FUNCTION_BLOCK FB_Double_drum
VAR_INPUT
	Lh_raw_depth:REAL; (*Raw left hand drum depth*)
	Rh_raw_depth:REAL; (*Raw right hand drum depth*)
	Lh_speed:REAL; (*Left drum speed in mm/s*)
	Rh_speed:REAL; (*Right drum speed in mm/s*)
	Tacho_speed:REAL; (*Tacho speed in mm/s*)
	Speed_ref:REAL; (*Speed reference output to drive in mm/s*)
	Lh_going_up:BOOL; (*Left conveyance moving in the upward direction (forward)*)
	Rh_going_up:BOOL; (*Right conveyance moving in the upward direction (forward)*)
	Lh_movement:BOOL; (*Movement detected on left drum since the brakes were last applied*)
	Rh_movement:BOOL; (*Movement detected on right drum since the brakes were last applied*)
	Enc_xcheck_dist:REAL; (*Allowed variation in the sum of the left and right raw depths since both clutches were put in or a winder reset*)
	Tacho_xcheck_abs:REAL; (*Allowed absolute difference between the tacho speed and encoder speed (added to Tacho_xcheck_percent)*)
	Tacho_xcheck_percent:REAL; (*Allowed percentage difference between the tacho speed and encoder speed (added to Tacho_xcheck_abs)*)
	Speed_ref_xcheck_abs:REAL; (*Allowed absolute difference between the speed reference (delayed) and the encoder speed (added to Speed_ref_xcheck_percent)*)
	Speed_ref_xcheck_percent:REAL; (*Allowed percentage difference between the speed reference (delayed) and the encoder speed (added to Speed_ref_xcheck_abs)*)
	System_response_time:REAL; (*Delay between giving the drive a reference and that speed being reached*)
	Speed_ave_scans:REAL;
END_VAR
VAR_OUTPUT
	Speed:REAL; (*Maximum speed between left and right encoders. Tacho is used if both encoders give zero speed.*)
	Movement:BOOL; (*Movement was detected on the left or right drum since the brakes were last applied*)
	Going_fwd:BOOL; (*The drums are moving in the forward direction*)
	Going_rev:BOOL; (*The drums are moving in the reverse direction*)
	Encoder_sum_xcheck:BOOL; (*The sum of the left and right raw depths has varied more than the allowed amount*)
	Lh_enc_vs_tacho_xcheck:BOOL; (*The difference between the tacho speed and left encoder speed was greater than the allowed amount*)
	Rh_enc_vs_tacho_xcheck:BOOL; (*The difference between the tacho speed and right encoder speed was greater than the allowed amount*)
	Speed_ref_xcheck:BOOL;(*The difference between the speed reference and encoder speed was greater than the allowed amount*)
END_VAR
VAR
	Speed_ref_delay_history:ARRAY[0..100]OF REAL;
	Speed_ref_delayed:REAL;
	System_response_scans:REAL;
	Rh_enc_tacho_diff:REAL;
	Lh_enc_tacho_diff:REAL;
	Speed_ref_diff:REAL;
	Encoder_sum:REAL;
	Required_encoder_sum:REAL;
	Window:REAL;
	F_TRIG_0: F_TRIG;
END_VAR

M_Double_drum_values();
M_Speed_crosschecks();
M_Depth_crosscheck();

METHOD M_Depth_crosscheck
VAR_INPUT
END_VAR
VAR_INST // added by the converter: edge detectors and wires of the graphical bodies
    _w1, _w2 : REAL;
END_VAR
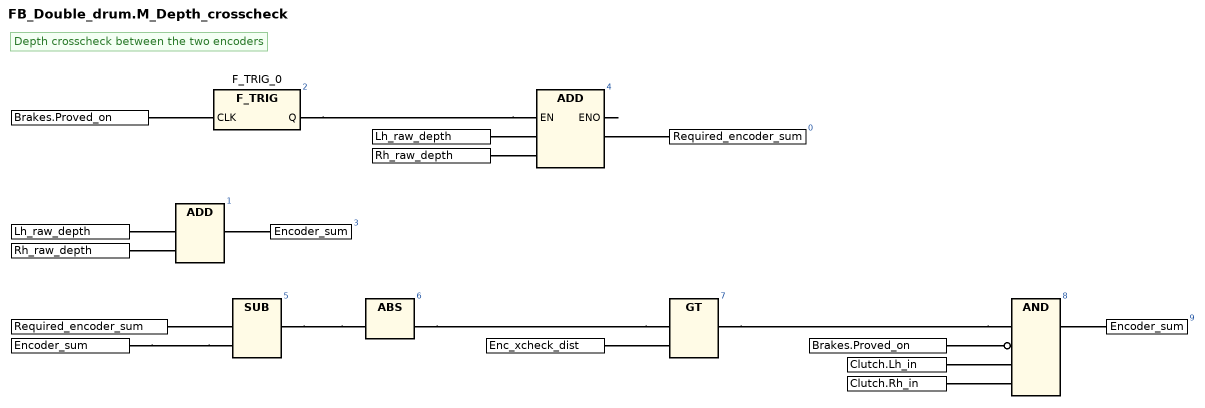
Required_encoder_sum := _w1;
_w2 := Lh_raw_depth + Rh_raw_depth;
// Depth crosscheck between the two encoders
F_TRIG_0(CLK := Brakes.Proved_on); // F_TRIG
Encoder_sum := _w2;
IF F_TRIG_0.Q THEN _w1 := Lh_raw_depth + Rh_raw_depth; END_IF
Encoder_sum := ABS(Required_encoder_sum - Encoder_sum) > Enc_xcheck_dist AND NOT Brakes.Proved_on AND Clutch.Lh_in AND Clutch.Rh_in;
END_METHOD

METHOD M_Double_drum_values
VAR_INPUT
END_VAR
VAR_INST // added by the converter: edge detectors and wires of the graphical bodies
    _w1, _w2, _w3, _w4, _w8, _w9 : BOOL;
    _w5, _w7 : REAL;
    _w6 : ANY;
END_VAR
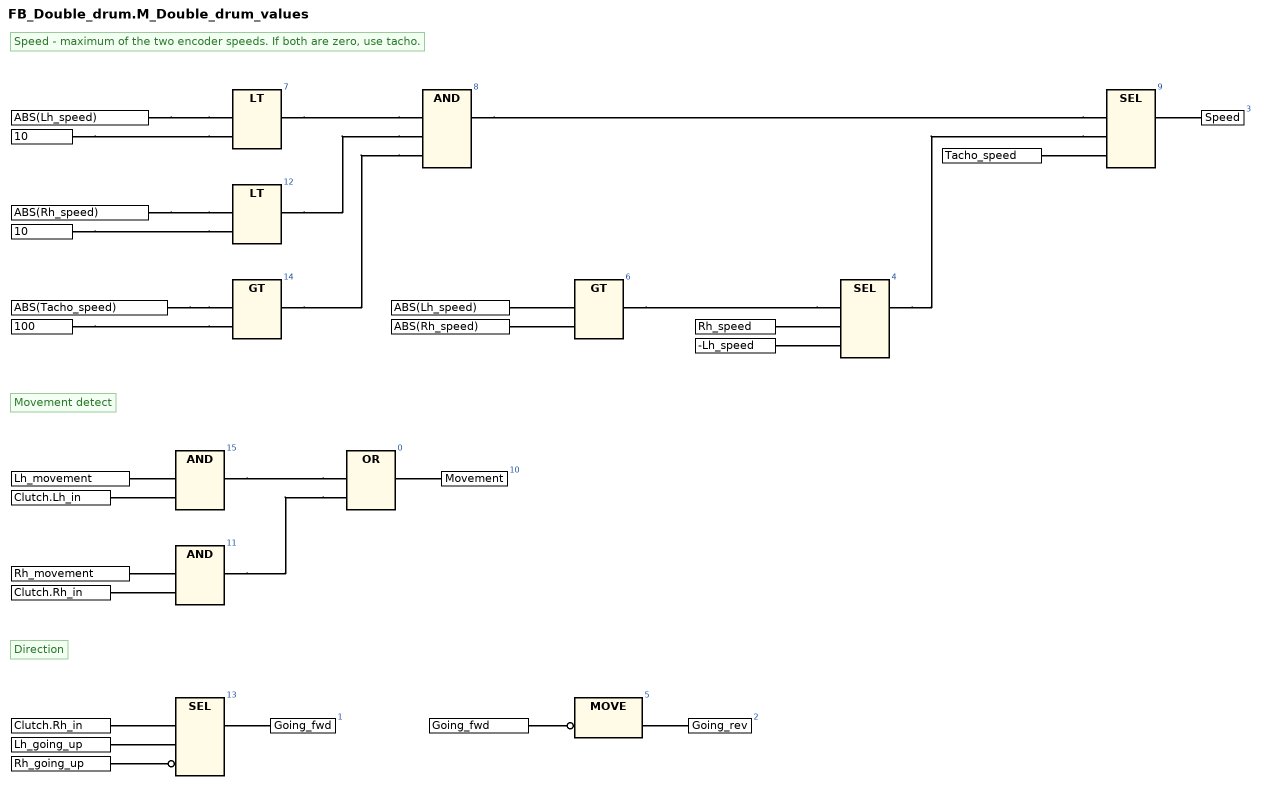
Going_fwd := _w3;
Going_rev := _w4;
Speed := _w5;
_w7 := SEL(_w6, Rh_speed, -Lh_speed);
_w4 := NOT Going_fwd;
_w6 := (ABS(Lh_speed)) > (ABS(Rh_speed));
// Speed - maximum of the two encoder speeds. If both are zero, use tacho.
_w5 := SEL((ABS(Lh_speed)) < 10 AND _w8 AND _w9, _w7, Tacho_speed);
Movement := _w1 OR _w2;
_w2 := Rh_movement AND Clutch.Rh_in;
_w8 := (ABS(Rh_speed)) < 10;
// Direction
_w3 := SEL(Clutch.Rh_in, Lh_going_up, NOT Rh_going_up);
_w9 := (ABS(Tacho_speed)) > 100;
// Movement detect
_w1 := Lh_movement AND Clutch.Lh_in;
END_METHOD

METHOD M_Speed_crosschecks
VAR_INPUT
END_VAR
VAR
	fbGetCurTaskIdx  : GETCURTASKINDEX;
	nIndex : DINT;
	nUpper : DINT;
	nLower : DINT;
END_VAR
{warning 'TODO: CycleTime here is implicitly converted from UDINT to REAL causing possible data loss.'}
{warning 'TODO: Ive re-written ROL_ARINT, please check @Bret'}
System_response_scans := System_response_time / _TaskInfo[fbGetCurTaskIdx.index].CycleTime;

(* Delay the speed reference to cater for the system response time *)	
//ROL_ARINT(1, Speed_ref_delay_history);

nUpper := UPPER_BOUND(Speed_ref_delay_history, 1);
nIndex := nUpper;

FOR nLower := LOWER_BOUND(Speed_ref_delay_history, 1) TO nUpper DO
	Speed_ref_delay_history[nIndex+1] := Speed_ref_delay_history[nIndex];
	nIndex := nIndex-1;
END_FOR
Speed_ref_delay_history[0] := Speed_ref;
Speed_ref_delayed := Speed_ref_delay_history[System_response_scans];

(* Now crosscheck the speeds. The speed reference will be used as the benchmark because it is the only one guaranteed to be correct. *)
(* The various speed values must agree within a percentage plus a fixed value for low speeds *)

Window := ABS(Speed_ref_delayed) * Tacho_xcheck_percent / 100.0 + Tacho_xcheck_abs;

(* Left encoder vs tacho crosscheck *)
Lh_enc_vs_tacho_xcheck := 0;
IF  Clutch.Lh_in THEN
	Lh_enc_tacho_diff := -Lh_speed - Tacho_speed;
	IF ABS(Lh_enc_tacho_diff) > Window THEN
		Lh_enc_vs_tacho_xcheck := 1;
	END_IF;
END_IF;

(* Right encoder vs tacho crosscheck *)
Rh_enc_vs_tacho_xcheck := 0;
IF Clutch.Rh_in THEN
	Rh_enc_tacho_diff := Rh_speed - Tacho_speed;
	IF ABS(Rh_enc_tacho_diff) > Window THEN
		Rh_enc_vs_tacho_xcheck := 1;
	END_IF;
END_IF;

(* Speed reference vs tacho crosscheck, i.e. speed reference not followed *)

Window := ABS(Speed_ref_delayed) * Speed_ref_xcheck_percent / 100.0 + Speed_ref_xcheck_abs;

Speed_ref_xcheck := 0;
Speed_ref_diff := Speed_ref_delayed - Tacho_speed;
IF ABS(Speed_ref_diff) > Window AND Safety.Sc1 THEN
	Speed_ref_xcheck := 1;
END_IF;
END_METHOD

END_FUNCTION_BLOCK

(* stored: Version 1.1.0.1, ProductVersion 3.1.4024.0
   POU FB_Double_drum: Id {15181611-30f7-4610-a263-4784b55c7bdf}, SpecialFunc None
   Method M_Depth_crosscheck: Id {bb7dfb9b-988e-4bc8-8c75-807a7ec7cd6f}
   Method M_Double_drum_values: Id {075d2d44-2c09-4e1b-8ea3-fb6f3465e061}
   Method M_Speed_crosschecks: Id {aee97c59-0506-4c16-8ea0-2deb56421f3a} *)
